FUNCTION_BLOCK ABSTRACT VisionHardwareNode EXTENDS HardwareNode IMPLEMENTS I_PreCheckedNode
VAR
	preExecutionCheckExtension : PreExecutionCheckExtension('precheck', THIS^);
END_VAR

METHOD PUBLIC Execute
IF NOT preExecutionCheckExtension.Check() THEN
	RETURN;
END_IF

SUPER^.Execute();
END_METHOD

METHOD PUBLIC ABSTRACT PreExecutionCheck
VAR_INPUT
	Check : I_PreExecutionChecks;
END_VAR
END_METHOD

END_FUNCTION_BLOCK

(* stored: Version 1.1.0.1, ProductVersion 3.1.4024.15
   POU VisionHardwareNode: Id {a5c48450-cc66-05c5-13da-5def0042a68e}, SpecialFunc None
   Method Execute: Id {f13616c6-9814-0efb-2103-ecbd257df9d3}
   Method PreExecutionCheck: Id {1075c372-f025-029e-0398-fe3c416da17f} *)
